// TIA Portal V19 export
DATA_BLOCK "Config"   // DB153
// stored: MemoryReserve 100, Namespace Unit.Em0
   VAR
      em { ExternalWritable := 'False'} : "LAF_typeEmConfiguration";   // Configuration of EM Parameters
   END_VAR
BEGIN
   em.referenceDesignator.parent := WSTRING#'Unit';
   em.referenceDesignator.relative := WSTRING#'EM0';
END_DATA_BLOCK
